FUNCTION Convert_LINT_TO_UINT : Hresult
VAR_INPUT
	in : LINT;
	out : REFERENCE TO UINT;
END_VAR
VAR
	converted : UINT;
END_VAR
VAR CONSTANT
	INCOMPATIBLE : HRESULT := 16#9811070E;
END_VAR

converted := LINT_TO_UINT(in);

IF (UINT_TO_LINT(converted) <> in) THEN
	Convert_LINT_TO_UINT := INCOMPATIBLE;
	RETURN;
END_IF

out := converted;

END_FUNCTION

(* stored: Version 1.1.0.1, ProductVersion 3.1.4024.12
   POU Convert_LINT_TO_UINT: Id {03c43add-ca02-496f-a917-1d9cf6e2ccd2}, SpecialFunc None *)
